(* Single tank with LimitSwitchLow (piLsLow) and LimitSwitchHigh (piLsHigh)
| using this function when it have INDEPENDENT Measure weight
*)
FUNCTION_BLOCK FB_SingleTankV1 EXTENDS FB_SingleTank
VAR
	bAllowInMaterial : BOOL;
	bAllowOutMaterial : BOOL;
	lrLimitMinWeight : LREAL;
	lrLimitMaxWeight : LREAL;
	lrWeightWithdraw : LREAL; 		// weight withdraw Request 
	bEnoughWithdraw : BOOL;
	lrWeight : LREAL;
END_VAR

bAllowInMaterial := lrWeight < lrLimitMaxWeight
						AND NOT piLsHigh.In;
						
bAllowOutMaterial := lrWeight > lrLimitMinWeight
						AND piLslow.In;
bEnoughWithdraw := lrWeight > (lrWeightWithdraw + lrLimitMinWeight);
SUPER^();

PROPERTY AllowIn : Reference to bool
GET
AllowIn ref= bAllowInMaterial;
END_GET
END_PROPERTY

(*
| Check the minimum condition  (lrWeight > lrLimitMinWeight
								AND piLslow.In;)
*)
PROPERTY AllowOut : REFERENCE TO BOOL
GET
AllowOut ref= bAllowOutMaterial;
END_GET
END_PROPERTY

(*
|Check enough weight to withdraw
*)
PROPERTY EnoughWithdraw : reference to bool
GET
EnoughWithdraw ref= bEnoughWithdraw;
END_GET
END_PROPERTY

PROPERTY LimitMaxWeight : LREAL
GET
LimitMaxWeight := lrLimitMaxWeight;
END_GET
SET
lrLimitMaxWeight := LimitMaxWeight;
END_SET
END_PROPERTY

PROPERTY LimitMinWeight : LREAL
GET
LimitMinWeight := lrLimitMinWeight;
END_GET
SET
lrLimitMinWeight := LimitMinWeight;
END_SET
END_PROPERTY

PROPERTY Weight : lreal
GET
Weight := lrWeight;
END_GET
SET
lrWeight := Weight;
END_SET
END_PROPERTY

PROPERTY WeightWithdraw : lreal
GET
WeightWithdraw := lrWeightWithdraw;
END_GET
SET
lrWeightWithdraw := WeightWithdraw;
END_SET
END_PROPERTY

END_FUNCTION_BLOCK

(* stored: Version 1.1.0.1, ProductVersion 3.1.4024.12
   POU FB_SingleTankV1: Id {3c3c8172-9c8e-4f0e-8bd8-ee41f1a2ec87}, SpecialFunc None
   Property AllowIn: Id {a5d1e9f2-1d23-4794-9392-8644ad8ab554}
   Get Get: Id {4611aad3-ae04-417a-8e61-b72d52a0c4c9}
   Property AllowOut: Id {5d4e6ea0-55ba-4704-a525-66ba75ae4a85}
   Get Get: Id {fa245f39-09b8-4716-b89c-489ebbbd1034}
   Property EnoughWithdraw: Id {14d668ef-cb0c-48e5-a28f-b4a763b749af}
   Get Get: Id {72331470-823e-4389-a30c-fc5d641e0da2}
   Property LimitMaxWeight: Id {09fb551a-44f6-4d4c-a29c-9adbf53bc1cd}
   Get Get: Id {02401e58-0bb9-42a3-8fe1-495c415f6569}
   Set Set: Id {2848334a-9b22-45d2-ac30-3fd5e06e6022}
   Property LimitMinWeight: Id {92119500-b222-4856-9d65-fe07625525b9}
   Get Get: Id {67a0b6a7-533a-440e-a39d-a2e2b1939326}
   Set Set: Id {d4aabfd8-d758-407f-a9a5-9feeba1db405}
   Property Weight: Id {48882b1a-1508-4301-adb8-c089b6bbba6d}
   Get Get: Id {362c66b8-ca90-4246-a487-4309fe64b699}
   Set Set: Id {67a10c51-fa14-474d-96ee-72217c924e34}
   Property WeightWithdraw: Id {6d9ed7fc-1a86-4025-a41e-3fd4479388ad}
   Get Get: Id {1111ca0d-4b93-425c-9139-7bcae5615117}
   Set Set: Id {b23ab4a6-f158-435d-89cf-39a8467e5856} *)
